// TIA Portal V19 export
DATA_BLOCK "CoilHandling"   // DB42
// stored: InstanceOfName CoilHandling_FB, InstanceOfType FB
"CoilHandling_FB"
   // VAR_INPUT
   //    AreaInterface : "AreaInterface";
   //    ZSI : "udt_ZoneSafetyInterface";
   //    DataIn : Struct
   //       PbMaterialBkw : Bool;
   //       PbMaterialFwd : Bool;
   //       PbExtraLowSpeed : Bool;
   //       SensorMatPresence_Decoiler : Bool;
   //       SensorMatPresence_StraightEntry : Bool;
   //       SensorMatPresence_StraightExit : Bool;
   //       SensorMatPresence_JBPinchExit : Bool;
   //       PbCoilReady : Bool;
   //       PbProvino : Bool;
   //       Decoiler2_PosizioneRazza : Bool;
   //    END_STRUCT;
   //    CIn : Struct
   //       DecoilersHRot : "DecoilersHRot_Status";
   //       Decoiler1 : "Decoiler_Status";
   //       Decoiler2 : "Decoiler_Status";
   //       Peeler : "Peeler_Status";
   //       Straigtener : "Straightener_Status";
   //       JB : "JB_Status";
   //       MaterialCounter : Struct
   //          AlrPresence : Bool;
   //          WngPresence : Bool;
   //          Data : "MatCountData";
   //       END_STRUCT;
   //       Loop : Struct
   //          SystemOn : Bool;
   //          Enable_FWD : Bool;
   //          Enable_BWD : Bool;
   //          SynchroRunning : Bool;
   //          MaxLength_Reeached : Bool;
   //          VelocityOverride : Real;
   //       END_STRUCT;
   //       Downstream : Struct
   //          Aut : Bool;
   //          MaterialPresence_Entry : Bool;
   //          MaterialPresence : Bool;
   //          LineVelocity : LReal;
   //       END_STRUCT;
   //       MES : "Prod_Coil_Ctrl";
   //    END_STRUCT;
   //    Config : "CoilHandling_Config";
   //    "ThicknessCheck_HW_ID_DL-PN" : HW_SUBMODULE;
   //    ThicknessCheck_HW_ID_IL1000 : HW_SUBMODULE;
   //    ThicknessCheck_HW_ID_IL1050 : HW_SUBMODULE;
   // END_VAR
   // VAR_OUTPUT
   //    MachineInterface : "MachineInterface";
   //    COut : Struct
   //       Gen : Struct
   //          Material_STS : Int;
   //          MaterialPresence : Bool;
   //          MaterialMissing : Bool;
   //          NextEndOfMaterial : Bool;
   //          EmptyingConfirmed : Bool;
   //          ExtraLowSpeedSelection : Bool;
   //          SemiAutomatic : Bool;
   //          Production_Running : Bool;
   //          DecoilerInLineNumber : Int;
   //          CoilDiameter : Real;
   //       END_STRUCT;
   //       DecoilersHRot : "DecoilersHRot_Manager";
   //       DecoilerInLine : "Decoiler_Manager";
   //       DecoilerOutLine : "Decoiler_Manager";
   //       Decoiler1 : "Decoiler_Manager";
   //       Decoiler2 : "Decoiler_Manager";
   //       Peeler : "Peeler_Manager";
   //       Straightener : "Straightener_Manager";
   //       JB : "JB_Manager";
   //       Loop : Struct
   //          Stop : Bool;
   //          Synchro_Request : Bool;
   //          MaterialMiddlePos_Request : Bool;
   //       END_STRUCT;
   //       MES : Struct
   //          Deroga_Spessore_Errato { ExternalWritable := 'False'} : Bool;
   //          Spessore_Lamiera_Errato { ExternalWritable := 'False'} : Bool;
   //          Spessore_Lamiera_Sensore_Valore : Real;
   //          Spessore_Lamiera_Errore_Valore { ExternalWritable := 'False'} : Real;
   //          Provino_Eseguito : Bool;
   //       END_STRUCT;
   //    END_STRUCT;
   //    DataOut : Struct
   //       Lamp_CoilReady : Bool;
   //       Lamp_ExtraLowSpeed : Bool;
   //       Lamp_Provino : Bool;
   //    END_STRUCT;
   // END_VAR
   // VAR_IN_OUT
   //    Pers : "CoilHandling_Persistent";
   // END_VAR
   // VAR
   //    Alarm : Struct
   //       MaterialMissing : Bool;
   //       S_MatPresence_StraightExit_NotOFF : Bool;
   //       MatCounterAlrPresence : Bool;
   //       EndOfMaterial : Bool;
   //       TichnessCheck { ExternalAccessible := 'False'; ExternalVisible := 'False'; ExternalWritable := 'False'} : Struct
   //          Err_Sensor_Get_PN_IO : Bool;
   //          Err_Sensor_Rack : Bool;
   //          Err_Sensor_Value : Bool;
   //          ThicknessOutOfRange : Bool;
   //       END_STRUCT;
   //       MES : Struct
   //          STOP_Provino { ExternalAccessible := 'False'; ExternalVisible := 'False'; ExternalWritable := 'False'} : Bool;
   //          STOP_Taglio_Fine_Ordini { ExternalAccessible := 'False'; ExternalVisible := 'False'; ExternalWritable := 'False'} : Bool;
   //          STOP_Manca_Dati_AspoInLinea { ExternalAccessible := 'False'; ExternalVisible := 'False'; ExternalWritable := 'False'} : Bool;
   //          STOP_FineTurno { ExternalAccessible := 'False'; ExternalVisible := 'False'; ExternalWritable := 'False'} : Bool;
   //          STOP_ControlloQualita { ExternalAccessible := 'False'; ExternalVisible := 'False'; ExternalWritable := 'False'} : Bool;
   //       END_STRUCT;
   //    END_STRUCT;
   //    Warning : Struct
   //       NotAutReady : Bool;
   //       MatCounterWngPresence : Bool;
   //       EmptyingIsON : Bool;
   //       EndOfMaterial_StraightenetEntry : Bool;
   //       EndOfMaterial_StraightenetExit : Bool;
   //       EndOfCoilSequenceRunning : Bool;
   //       ExtraLowSpeedIsON : Bool;
   //       Decoiler2_RazzaNonInPosizione : Bool;
   //       StopInactivity : Bool;
   //       ThicnessCheck { ExternalAccessible := 'False'; ExternalVisible := 'False'; ExternalWritable := 'False'} : Struct
   //          SensorDisable : Bool;
   //          ThicknessOutOfRange : Bool;
   //          Err_Bypass : Bool;
   //       END_STRUCT;
   //       MES : Struct
   //          STOP_Manca_Dati_AspoInCarico : Bool;
   //       END_STRUCT;
   //    END_STRUCT;
   //    HMI : Struct
   //       B_ConfirmEmptying { ExternalAccessible := 'False'; ExternalVisible := 'False'; ExternalWritable := 'False'} : Bool;
   //       B_ConfirmEmptyingShow { ExternalAccessible := 'False'; ExternalVisible := 'False'; ExternalWritable := 'False'} : Bool;
   //       B_ConfirmEmptyingStatus : Bool;
   //       ThicknessControl : Struct
   //          Button_Exception : Bool;
   //          Button_Init : Bool;
   //          STATUS : Int;
   //       END_STRUCT;
   //    END_STRUCT;
   //    Ctrl : Struct
   //       Pause : Bool;
   //       Stop : Bool;
   //       Semiautomatic_MaterialFwd : Bool;
   //       Semiautomatic_MaterialBkw : Bool;
   //       EndOfCoil : Struct
   //          StraightRollEntry_Open : Bool;
   //          StraightRollExit_Open : Bool;
   //          StraightRollEntry_Close : Bool;
   //          StraightRollExit_Close : Bool;
   //          Straightener_Bwd : Bool;
   //          Straightener_Fwd : Bool;
   //          JB_Pinch_Open : Bool;
   //          JB_Pinch_Close : Bool;
   //          JB_Pinch_Fwd : Bool;
   //          JB_Cut_Rest : Bool;
   //          JB_Cut_Work : Bool;
   //          JB_Welder_Open : Bool;
   //          TargetPosMat_StraightEmpty : LReal;
   //          TargetPosMat_TailCutExe : LReal;
   //          TargetPosMat_JunctionExe : LReal;
   //          ChangeCoilExe : Bool;
   //          Decoiler_Fwd : Bool;
   //       END_STRUCT;
   //    END_STRUCT;
   //    Sts : Struct
   //       FeedStandstill : Bool;
   //       AlarmsPresence : Bool;
   //       WarningsPresence : Bool;
   //       EnableCycleStopProgrammed : Bool;
   //       MaterialFwdEnable : Bool;
   //       MaterialBkwEnable : Bool;
   //       CumulativeMaterialFwdRequest : Bool;
   //       Semiautomatic : Bool;
   //       ExtraLowSpeedSelectionPB : Bool;
   //       ExtraLowSpeedSelection : Bool;
   //       STOP_Feed_by_MES : Bool;
   //       STOP_CoilChange_By_MES : Bool;
   //       STOP_Inactivity : Bool;
   //       DecoilerInLine : "Decoiler_Status";
   //       DecoilerOutOfLine : "Decoiler_Status";
   //       EndOfCoil : Struct
   //          Status : Int;
   //          Cnd : Bool;
   //          Idle : Bool;
   //          EndOfSequence : Bool;
   //          PinchRoll_SpaceToStop : LReal;
   //          PosMat_AtEndMatPresence_StraightEnty : LReal;
   //          PosMat_AtEndMatPresence_StraightExit : LReal;
   //          MissingTargetPosMat_StraightEmpty : LReal;
   //          MissingToTargetPosMat_TailCutExe : LReal;
   //          StopPinchRoll_TargetPosMat_TailCutExe : Bool;
   //          Reached_TargetPosMat_TailCutExe : Bool;
   //          MissingToTargetPosMat_JunctionExe : LReal;
   //          StopPinchRoll_TargetPosMat_JunctionExe : Bool;
   //          Reached_TargetPosMat_JunctionExe : Bool;
   //       END_STRUCT;
   //       LoopSynchro : Struct
   //          Phase1_A : Bool;
   //          Phase2_A : Bool;
   //          Phase1_B : Bool;
   //          Phase2_B : Bool;
   //       END_STRUCT;
   //       MaterialMoveSemiAut : Struct
   //          Bwd_Phase1 : Bool;
   //          Bwd_Phase1Cnd : Bool;
   //          Bwd_Phase2 : Bool;
   //          Bwd_Phase2Cnd : Bool;
   //          Bwd_Phase3 : Bool;
   //          Fwd_Phase1 : Bool;
   //          Fwd_Phase1Cnd : Bool;
   //          Fwd_Phase2 : Bool;
   //          Fwd_Phase2Cnd : Bool;
   //          Fwd_Phase3 : Bool;
   //       END_STRUCT;
   //       MaterialMoveAut : Struct
   //          Fwd_Phase1 : Bool;
   //          Fwd_Phase1Cnd : Bool;
   //          Fwd_Phase2 : Bool;
   //          Fwd_Phase2Cnd : Bool;
   //          Fwd_Phase3 : Bool;
   //       END_STRUCT;
   //    END_STRUCT;
   //    MatPresence_Decoiler : "DelayOnOff_R";
   //    MatPresence_StraightEntry : "DelayOnOff_R";
   //    MatPresence_StraightExit : "DelayOnOff_R";
   //    MatPresence_JBPinchExit : "DelayOnOff_R";
   //    Coil_LooseWrap : "CoilCheckLooseWrap";
   //    ThicknessCheck { S7_SetPoint := 'True'} : "ThicknessCheck_FB";
   //    CoilHandling_MES { S7_SetPoint := 'True'} : "CoilHandling_MES_FB";
   //    TON_Emptying : TON_TIME;
   //    TON_DecoilerNotMovingBkw : TON_TIME;
   //    TON_PinchrollFwd : TON_TIME;
   //    TON_StraightnerBwd : TON_TIME;
   //    TON_StraightnerFwd : TON_TIME;
   //    TON_SemiautoOFF : TON_TIME;
   //    TON_AutDisableAxes : TON_TIME;
   //    TON_StopInactivity : TON_TIME;
   //    AUX : Struct
   //       S_MatPresence_StraightEntry : Bool;
   //       S_MatPresence_StraightExit : Bool;
   //       PbMaterialFwd : Bool;
   //       PbMaterialBkw : Bool;
   //       PbExtraLowSpeed : Bool;
   //       ButtonForceLoopMiddle : Bool;
   //       PbCoilLoaded : Bool;
   //       StopLoop { ExternalAccessible := 'False'; ExternalVisible := 'False'; ExternalWritable := 'False'} : Bool;
   //    END_STRUCT;
   // END_VAR
BEGIN
END_DATA_BLOCK
